// TIA Portal V20 export
VAR_GLOBAL   // PLC tag table "Unit1Em3_Servo"
   "BA030AZSBK01.03" AT %I1000.3 : Bool;   // COMPENSATOR LIMIT SENSOR(-)
   "BA030AZSBK01.04" AT %I1000.4 : Bool;   // COMPENSATOR LIMIT SENSOR(+)
   "BA030AZSBK01.13" AT %I1001.3 : Bool;   // COMPENSATOR HOME SENSOR
END_VAR
